(*

.. <legal notes>

legal notes
=================
| SPDX-FileCopyrightText: © 2025 Oleksandr Tiutyk <trofimich@gmail.com>
| SPDX-License-Identifier: LGPL-3.0-only
| For details check: LGPL-3.0-only_

.. _LGPL-3.0-only: https://www.gnu.org/licenses/lgpl-3.0.en.html

.. </legal notes>

*)

{attribute 'no_explicit_call' := 'Direct call is not allowed'} 
FUNCTION_BLOCK FileContentTaskQueue EXTENDS TOF_Tasks.Task
VAR
	_FileManagerClassName : STRING := __POUNAME();
	
	_Open : Tc2_System.FB_FileOpen;
	_Close : Tc2_System.FB_FileClose;
	
	_Starting : BOOL;
		
	_TaskQueue : TOF_Tasks.TaskQueue;
END_VAR

{attribute 'monitoring' := 'call'}
{attribute 'OPC.UA.DA.Property' := '1'}
{attribute 'OPC.UA.DA' := '1'}
PROPERTY AmsNetId : Tc2_System.T_AmsNetID
GET
AmsNetId := _Open.sNetId;
END_GET
SET
_Open.sNetId := AmsNetId;
_Close.sNetId := AmsNetId;
END_SET
END_PROPERTY

{attribute 'monitoring' := 'call'}
PROPERTY ClassName : STRING
GET
ClassName := _FileManagerClassName;
END_GET
END_PROPERTY

METHOD FINAL ClearTasks
_TaskQueue.Clear();
END_METHOD

METHOD Enqueue
VAR_INPUT
	fileHandleTask : IFileContentTask; 
	deleteOnFinishOrClear : BOOL := FALSE;
END_VAR
IF fileHandleTask <> 0 THEN
	fileHandleTask.SetFileOpen(_Open);
	
	_TaskQueue.Enqueue(fileHandleTask, deleteOnFinishOrClear);
END_IF
END_METHOD

METHOD PRIVATE fileClose
_Close(bExecute := TRUE, hFile := _Open.hFile);
_Open(bExecute := FALSE);
	
TOF_Core.LogManager.TryLogMessage(WideStringHelper.ConcatStrings255("Attempt to close file '", TO_WSTRING(_Open.sPathName), "'"), LOG_CATEGORY.INFORMATION, "FileManager", "FileManager.FileCloseAttempt");
END_METHOD

{attribute 'monitoring' := 'call'}
PROPERTY FINAL FileHandle : UINT
GET
FileHandle := _Open.hFile;
END_GET
END_PROPERTY

METHOD PRIVATE fileOpen
_Close(bExecute := FALSE);
_Open(bExecute := TRUE);
	
TOF_Core.LogManager.TryLogMessage(WideStringHelper.ConcatStrings255("Attempt to open file '", TO_WSTRING(_Open.sPathName), "'"), LOG_CATEGORY.INFORMATION, "FileManager", "FileManager.FileOpenAttempt");
END_METHOD

{attribute 'monitoring' := 'call'}
PROPERTY FilePath : Tc2_System.T_MaxString
GET
FilePath := _Open.sPathName;
END_GET
SET
_Open.sPathName := FilePath;
END_SET
END_PROPERTY

{attribute 'monitoring' := 'call'}
// use Tc2_System.Global_Variables.FOPEN_MODEXXX
PROPERTY ModeFlags : DWORD
GET
ModeFlags := _Open.nMode;
END_GET
SET
_Open.nMode := ModeFlags;
END_SET
END_PROPERTY

{attribute 'monitoring' := 'call'}
PROPERTY NamespaceName : STRING
GET
NamespaceName := CurrentNamespace.Name;
END_GET
END_PROPERTY

METHOD PROTECTED OnCancel
_TaskQueue.Cancel();

fileClose();
END_METHOD

METHOD PROTECTED OnFault
fileClose();
END_METHOD

METHOD PROTECTED OnRunning 
VAR_INPUT
	startRequest : BOOL;
END_VAR
VAR_OUTPUT
	state : TASK_RUNNING_STATE;
END_VAR
VAR
	memberNotSpecifiedException : DataMemberNotSpecifiedException;
	deleteDirectoryException : TOF_Core.StandardException;
	invalidPathException : InvalidPathException;	

	pathErrorMessage : WSTRING(255);
	errorMessageBuilder : TOF_Core.WideStringBuilder;	
END_VAR
IF startRequest THEN
	IF TOF_Core.StringHelper.IsNullOrWhiteSpace(_Open.sPathName) THEN
		memberNotSpecifiedException.Throw(NameSpacename, ClassName, __POUNAME(), __POSITION(), 'FilePath');
	END_IF

	fileOpen();
	
	_Starting := TRUE;
	
	RETURN;
ELSE		
	IF _Starting THEN
		_Close();
		_Open();
		
		IF _Open.bError THEN
			errorMessageBuilder
				.AppendString("Error while open file '")
				.Append(_Open.sPathName)
				.AppendString("'");
		
			deleteDirectoryException.Throw(NamespaceName, ClassName, __POUNAME(), __POSITION(), errorMessageBuilder.ToString255());		
		END_IF
		
		IF _Open.bBusy THEN
			RETURN;
		END_IF

		_Starting := FALSE;
		
		_TaskQueue.Start();
	ELSE
		_TaskQueue.Execute(); 
	END_IF
END_IF

IF NOT _TaskQueue.Busy THEN
	IF _TaskQueue.Done THEN	
		state := TASK_RUNNING_STATE.DONE;
	ELSIF _TaskQueue.Aborted THEN
		state := TASK_RUNNING_STATE.ABORTED;
	END_IF	

	fileClose();
END_IF
END_METHOD

{attribute 'monitoring' := 'call'}
PROPERTY PathType : Tc2_System.E_OpenPath
GET
PathType := _Open.ePath;
END_GET
SET
_Open.ePath := PathType;
END_SET
END_PROPERTY

{attribute 'monitoring' := 'call'}
PROPERTY FINAL PendingTaskCount : DINT
GET
PendingTaskCount := _TaskQueue.PendingTaskCount;
END_GET
END_PROPERTY

{attribute 'monitoring' := 'call'}
PROPERTY Size : ULINT
GET
Size := XSIZEOF(THIS^);
END_GET
END_PROPERTY

{attribute 'monitoring' := 'call'}
{attribute 'OPC.UA.DA.Property' := '1'}
{attribute 'OPC.UA.DA' := '1'}
PROPERTY Timeout : TIME
GET
Timeout := _Open.tTimeout;
END_GET
SET
_Open.tTimeout := Timeout;
_Close.tTimeout := Timeout;
END_SET
END_PROPERTY

END_FUNCTION_BLOCK

(* stored: Version 1.1.0.1
   POU FileContentTaskQueue: Id {bc2051e9-92a1-4c8e-a38d-beb02683c33f}, SpecialFunc None
   Folder Inputs: Id {bfacd55a-3afa-44c2-84dc-abf547a00bf3}
   Folder Outputs: Id {9ba5e1c6-a771-4234-bb21-c0bdd9c29447}
   Folder Overriden members: Id {b5902f7c-0b68-468a-aed6-ab0827abdd52}
   Folder Service memebers: Id {10603918-70f1-4abe-9de6-dff33e7d7d98}
   Property AmsNetId: Id {1c569c82-f0ee-422a-ab1a-6efc60d4b20b}
   Get Get: Id {a36a3a86-9c70-41e1-acd3-9b400a782ee7}
   Set Set: Id {5dd72bd3-ffb7-47df-9468-d7385af74eaf}
   Property ClassName: Id {7dde5df2-bee6-469e-a34d-e38f282681a9}
   Get Get: Id {d478f9e9-291b-4ed2-a175-f912be663022}
   Method ClearTasks: Id {8c96f5d2-116d-4613-b8ca-9482f7ab04c1}
   Method Enqueue: Id {6d338e28-e90a-4f1d-be55-6a823f742ef9}
   Method fileClose: Id {023ab949-b21b-4f26-9304-fdefb517b6cf}
   Property FileHandle: Id {d400f36f-4560-4321-9301-560723b5321c}
   Get Get: Id {af4ff15c-e163-44de-a875-054227fd820a}
   Method fileOpen: Id {c22dda38-9bc7-4659-be27-9091bae2b4a7}
   Property FilePath: Id {f39c82db-1dee-4ac8-b085-ad0d066c8468}
   Get Get: Id {c797c652-63c0-4561-b531-110a18c85ac4}
   Set Set: Id {b19d239b-2520-4cac-89cd-a80f2163f042}
   Property ModeFlags: Id {eab34e5a-e16f-430d-90f0-029e4eb57eb1}
   Get Get: Id {cebcc8dc-c629-4eab-8dfa-12a6c42e8047}
   Set Set: Id {f58cc275-9775-4af7-bb51-396283f88ce4}
   Property NamespaceName: Id {7b18bdc5-244f-4cb6-a69d-ff82980ef6e3}
   Get Get: Id {d8cd630c-d3f9-42c5-ba22-d2cd3c67dc04}
   Method OnCancel: Id {7771e8ba-0d52-4fbe-9407-bb22f236fecd}
   Method OnFault: Id {73768d9b-a52e-4b50-963d-d1ba76459290}
   Method OnRunning: Id {96e54c5c-06cb-46ed-bca0-9f0bd8bfc283}
   Property PathType: Id {cbd2448b-000c-4456-acbb-370bcc431295}
   Get Get: Id {4fd9cd50-b095-453b-aa33-3b46437fbccc}
   Set Set: Id {c88e846f-0d0c-469c-b204-0549d3f33d59}
   Property PendingTaskCount: Id {d108cb5f-99bc-48a9-ab2b-56da3b0f948f}
   Get Get: Id {32398972-9e42-46b6-a8d9-ee3d9bdb5dc1}
   Property Size: Id {aa575a10-da54-44bb-a1d2-ac20af742a7b}
   Get Get: Id {46726470-3c47-4383-bc77-fbfb39b4cbc0}
   Property Timeout: Id {8b8e24f2-ac37-4ffd-b14b-41645bab1c20}
   Get Get: Id {4943b545-4a96-4943-8f75-27394e4b849b}
   Set Set: Id {b3a6fe7d-0099-4655-a68b-17e02235542c} *)
